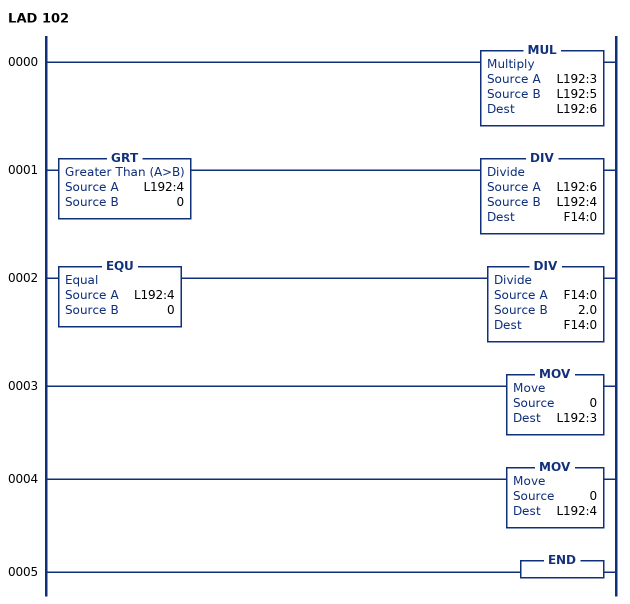
% Rung: 0 %
SOR MUL L192:3 L192:5 L192:6 EOR
% Rung: 1 %
SOR GRT L192:4 0 DIV L192:6 L192:4 F14:0 EOR
% Rung: 2 %
SOR EQU L192:4 0 DIV F14:0 2.0 F14:0 EOR
% Rung: 3 %
SOR MOV 0 L192:3 EOR
% Rung: 4 %
SOR MOV 0 L192:4 EOR
% Rung: 5 %
SOR END EOR

LADDER 103
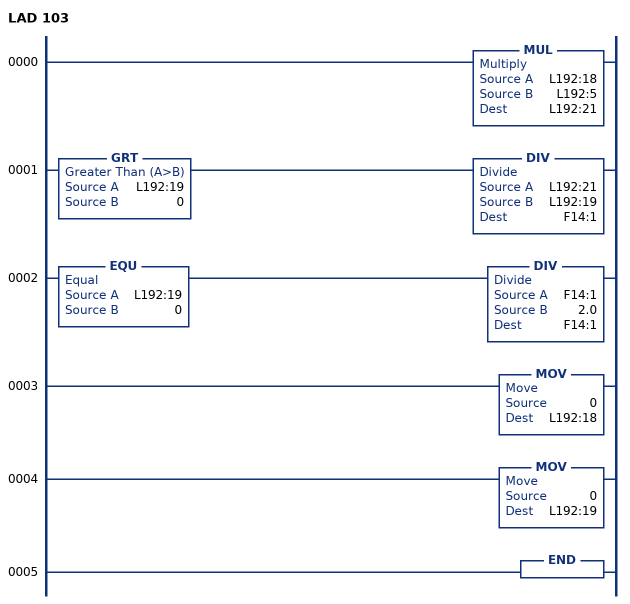
% Rung: 0 %
SOR MUL L192:18 L192:5 L192:21 EOR
% Rung: 1 %
SOR GRT L192:19 0 DIV L192:21 L192:19 F14:1 EOR
% Rung: 2 %
SOR EQU L192:19 0 DIV F14:1 2.0 F14:1 EOR
% Rung: 3 %
SOR MOV 0 L192:18 EOR
% Rung: 4 %
SOR MOV 0 L192:19 EOR
% Rung: 5 %
SOR END EOR

LADDER 104
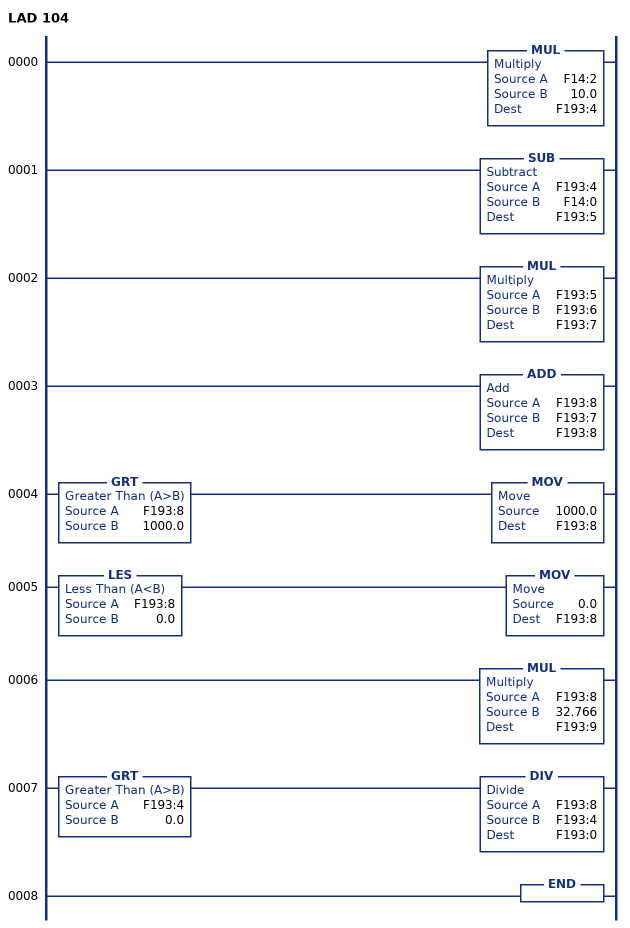
% Rung: 0 %
SOR MUL F14:2 10.0 F193:4 EOR
% Rung: 1 %
SOR SUB F193:4 F14:0 F193:5 EOR
% Rung: 2 %
SOR MUL F193:5 F193:6 F193:7 EOR
% Rung: 3 %
SOR ADD F193:8 F193:7 F193:8 EOR
% Rung: 4 %
SOR GRT F193:8 1000.0 MOV 1000.0 F193:8 EOR
% Rung: 5 %
SOR LES F193:8 0.0 MOV 0.0 F193:8 EOR
% Rung: 6 %
SOR MUL F193:8 32.766 F193:9 EOR
% Rung: 7 %
SOR GRT F193:4 0.0 DIV F193:8 F193:4 F193:0 EOR
% Rung: 8 %
SOR END EOR

LADDER 105
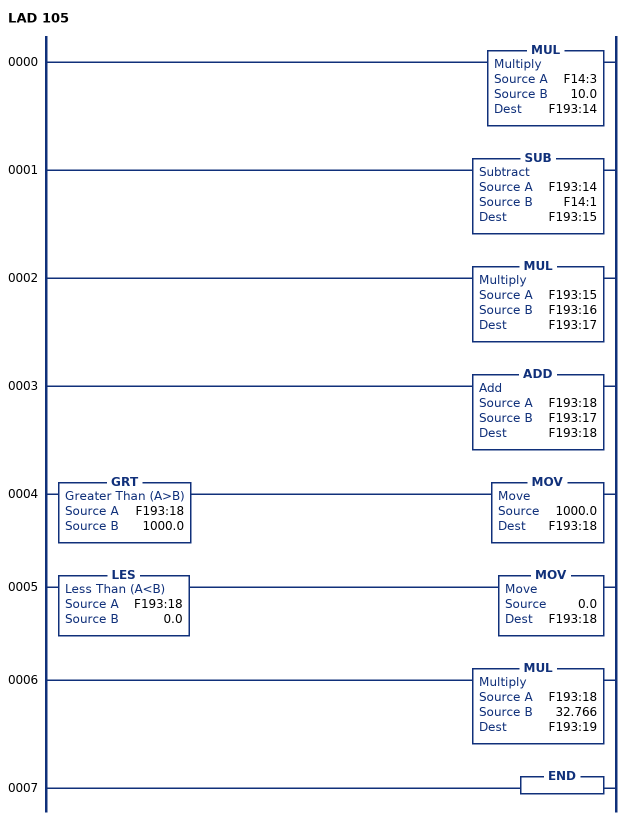
% Rung: 0 %
SOR MUL F14:3 10.0 F193:14 EOR
% Rung: 1 %
SOR SUB F193:14 F14:1 F193:15 EOR
% Rung: 2 %
SOR MUL F193:15 F193:16 F193:17 EOR
% Rung: 3 %
SOR ADD F193:18 F193:17 F193:18 EOR
% Rung: 4 %
SOR GRT F193:18 1000.0 MOV 1000.0 F193:18 EOR
% Rung: 5 %
SOR LES F193:18 0.0 MOV 0.0 F193:18 EOR
% Rung: 6 %
SOR MUL F193:18 32.766 F193:19 EOR
% Rung: 7 %
SOR END EOR

LADDER 110
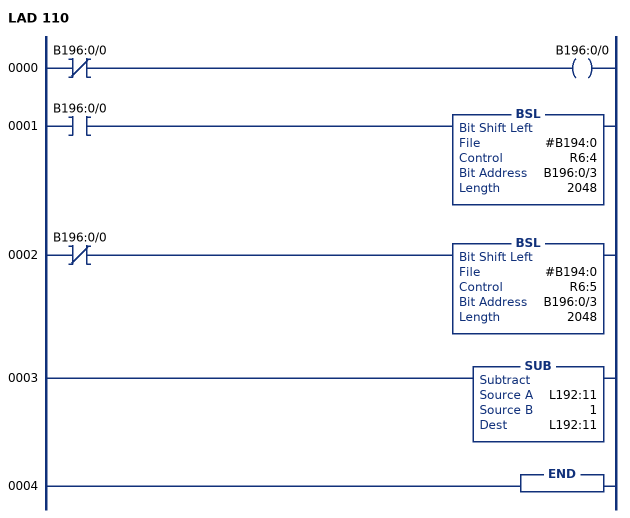
% Rung: 0 %
SOR XIO B196:0/0 OTE B196:0/0 EOR
% Rung: 1 %
SOR XIC B196:0/0 BSL #B194:0 R6:4 B196:0/3 2048 EOR
% Rung: 2 %
SOR XIO B196:0/0 BSL #B194:0 R6:5 B196:0/3 2048 EOR
% Rung: 3 %
SOR SUB L192:11 1 L192:11 EOR
% Rung: 4 %
SOR END EOR

LADDER 111
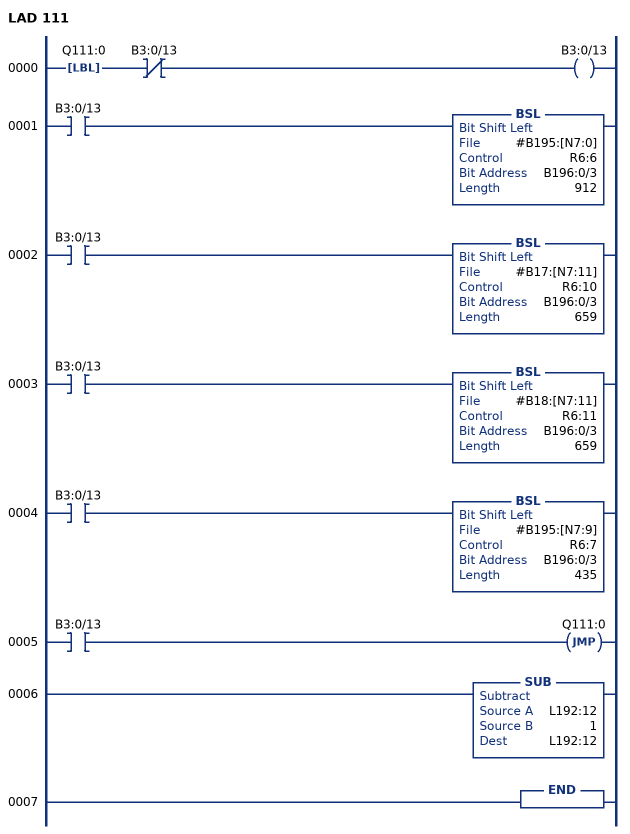
% Rung: 0 %
SOR LBL Q111:0 XIO B3:0/13 OTE B3:0/13 EOR
% Rung: 1 %
SOR XIC B3:0/13 BSL #B195:[N7:0] R6:6 B196:0/3 912 EOR
% Rung: 2 %
SOR XIC B3:0/13 BSL #B17:[N7:11] R6:10 B196:0/3 659 EOR
% Rung: 3 %
SOR XIC B3:0/13 BSL #B18:[N7:11] R6:11 B196:0/3 659 EOR
% Rung: 4 %
SOR XIC B3:0/13 BSL #B195:[N7:9] R6:7 B196:0/3 435 EOR
% Rung: 5 %
SOR XIC B3:0/13 JMP Q111:0 EOR
% Rung: 6 %
SOR SUB L192:12 1 L192:12 EOR
% Rung: 7 %
SOR END EOR

LADDER 122
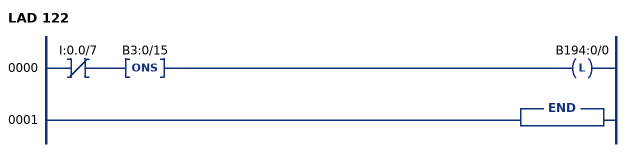
% Rung: 0 %
SOR XIO I:0.0/7 ONS B3:0/15 OTL B194:0/0 EOR
% Rung: 1 %
SOR END EOR

LADDER 125
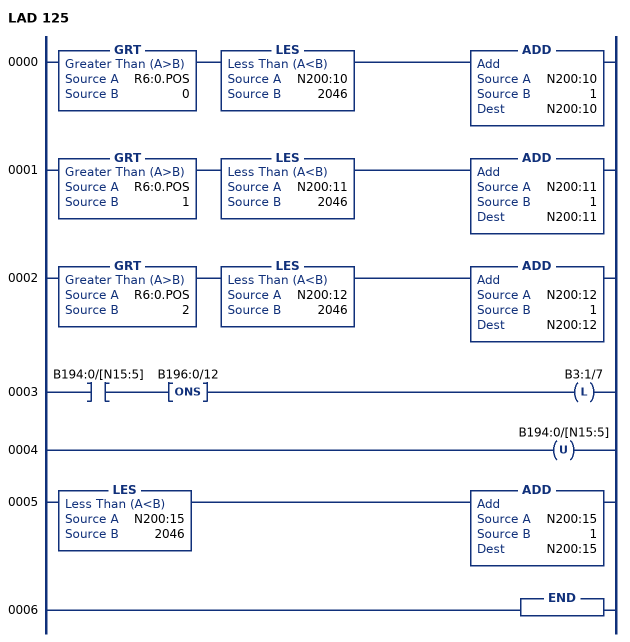
% Rung: 0 %
SOR GRT R6:0.POS 0 LES N200:10 2046 ADD N200:10 1 N200:10 EOR
% Rung: 1 %
SOR GRT R6:0.POS 1 LES N200:11 2046 ADD N200:11 1 N200:11 EOR
% Rung: 2 %
SOR GRT R6:0.POS 2 LES N200:12 2046 ADD N200:12 1 N200:12 EOR
% Rung: 3 %
SOR XIC B194:0/[N15:5] ONS B196:0/12 OTL B3:1/7 EOR
% Rung: 4 %
SOR OTU B194:0/[N15:5] EOR
% Rung: 5 %
SOR LES N200:15 2046 ADD N200:15 1 N200:15 EOR
% Rung: 6 %
SOR END EOR

LADDER 126
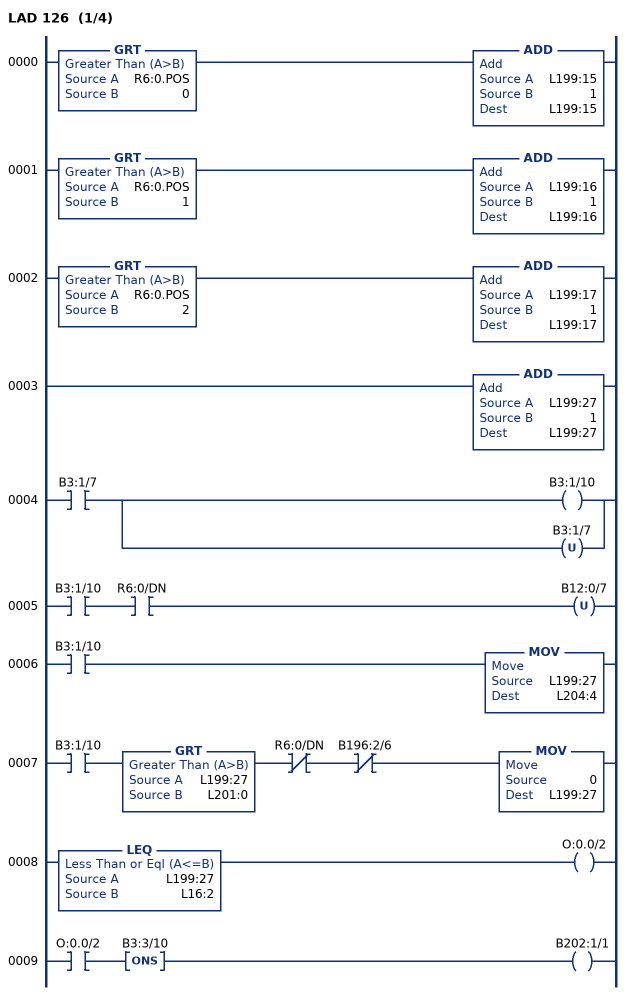
% Rung: 0 %
SOR GRT R6:0.POS 0 ADD L199:15 1 L199:15 EOR
% Rung: 1 %
SOR GRT R6:0.POS 1 ADD L199:16 1 L199:16 EOR
% Rung: 2 %
SOR GRT R6:0.POS 2 ADD L199:17 1 L199:17 EOR
% Rung: 3 %
SOR ADD L199:27 1 L199:27 EOR
% Rung: 4 %
SOR XIC B3:1/7 BST OTE B3:1/10 NXB OTU B3:1/7 BND EOR
% Rung: 5 %
SOR XIC B3:1/10 XIC R6:0/DN OTU B12:0/7 EOR
% Rung: 6 %
SOR XIC B3:1/10 MOV L199:27 L204:4 EOR
% Rung: 7 %
SOR XIC B3:1/10 GRT L199:27 L201:0 XIO R6:0/DN XIO B196:2/6 MOV 0 L199:27 EOR
% Rung: 8 %
SOR LEQ L199:27 L16:2 OTE O:0.0/2 EOR
% Rung: 9 %
SOR XIC O:0.0/2 ONS B3:3/10 OTE B202:1/1 EOR

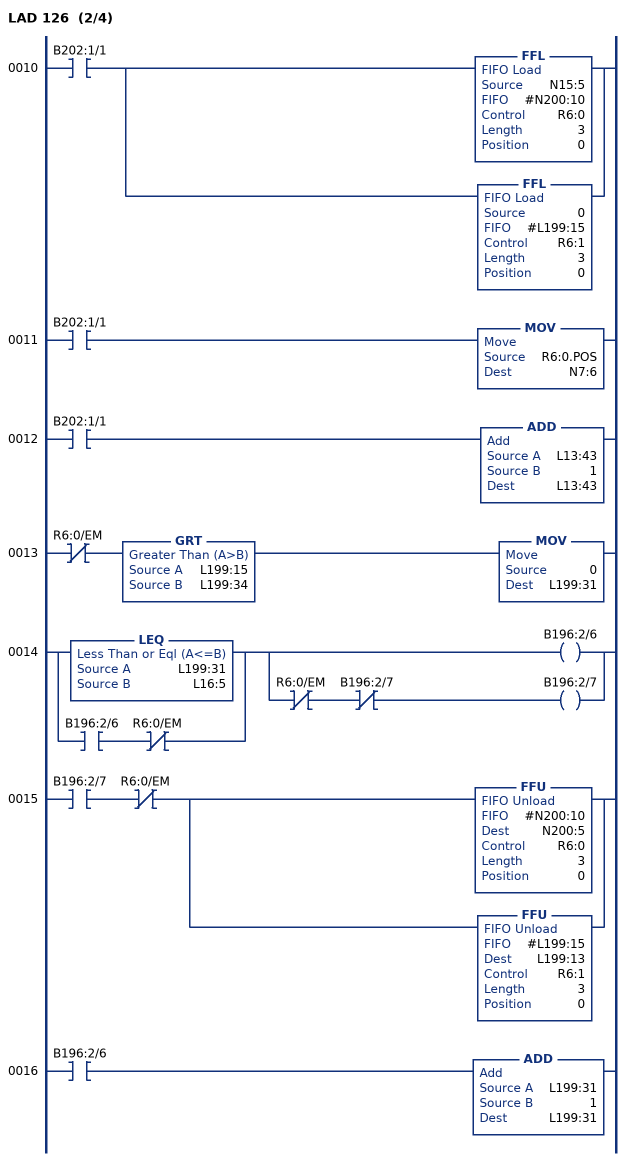
% Rung: 10 %
SOR XIC B202:1/1 BST FFL N15:5 #N200:10 R6:0 3 0 NXB FFL 0 #L199:15 R6:1 3 0 BND EOR
% Rung: 11 %
SOR XIC B202:1/1 MOV R6:0.POS N7:6 EOR
% Rung: 12 %
SOR XIC B202:1/1 ADD L13:43 1 L13:43 EOR
% Rung: 13 %
SOR XIO R6:0/EM GRT L199:15 L199:34 MOV 0 L199:31 EOR
% Rung: 14 %
SOR BST LEQ L199:31 L16:5 NXB XIC B196:2/6 XIO R6:0/EM BND BST OTE B196:2/6 NXB XIO R6:0/EM XIO B196:2/7 OTE B196:2/7 BND EOR
% Rung: 15 %
SOR XIC B196:2/7 XIO R6:0/EM BST FFU #N200:10 N200:5 R6:0 3 0 NXB FFU #L199:15 L199:13 R6:1 3 0 BND EOR
% Rung: 16 %
SOR XIC B196:2/6 ADD L199:31 1 L199:31 EOR

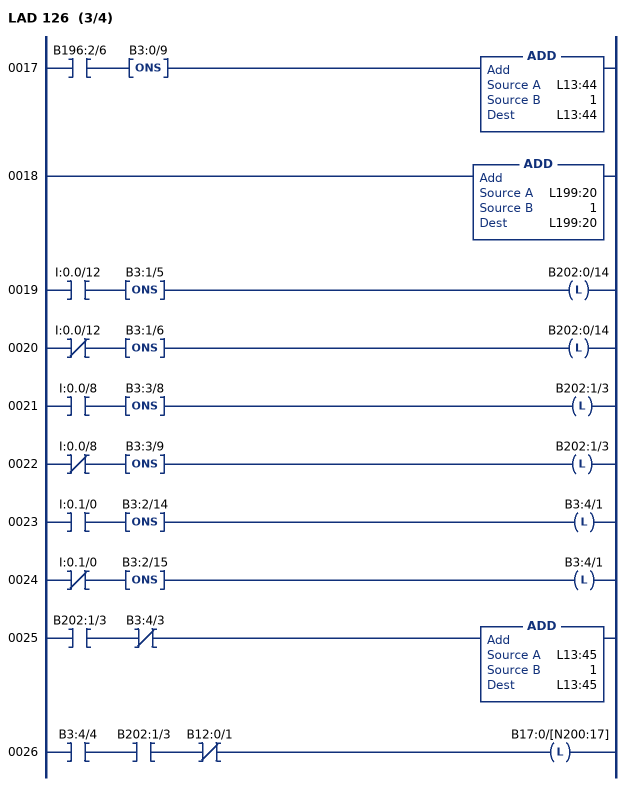
% Rung: 17 %
SOR XIC B196:2/6 ONS B3:0/9 ADD L13:44 1 L13:44 EOR
% Rung: 18 %
SOR ADD L199:20 1 L199:20 EOR
% Rung: 19 %
SOR XIC I:0.0/12 ONS B3:1/5 OTL B202:0/14 EOR
% Rung: 20 %
SOR XIO I:0.0/12 ONS B3:1/6 OTL B202:0/14 EOR
% Rung: 21 %
SOR XIC I:0.0/8 ONS B3:3/8 OTL B202:1/3 EOR
% Rung: 22 %
SOR XIO I:0.0/8 ONS B3:3/9 OTL B202:1/3 EOR
% Rung: 23 %
SOR XIC I:0.1/0 ONS B3:2/14 OTL B3:4/1 EOR
% Rung: 24 %
SOR XIO I:0.1/0 ONS B3:2/15 OTL B3:4/1 EOR
% Rung: 25 %
SOR XIC B202:1/3 XIO B3:4/3 ADD L13:45 1 L13:45 EOR
% Rung: 26 %
SOR XIC B3:4/4 XIC B202:1/3 XIO B12:0/1 OTL B17:0/[N200:17] EOR

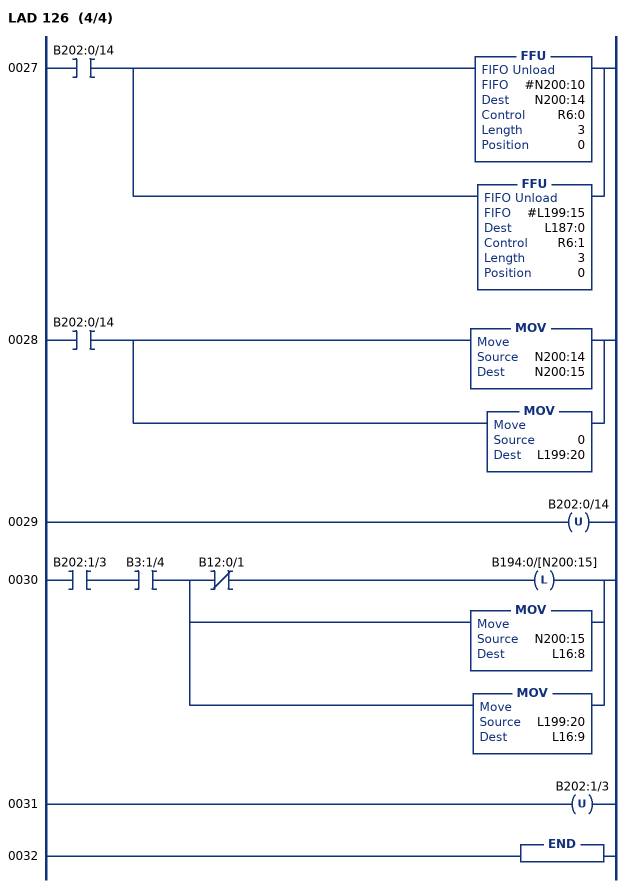
% Rung: 27 %
SOR XIC B202:0/14 BST FFU #N200:10 N200:14 R6:0 3 0 NXB FFU #L199:15 L187:0 R6:1 3 0 BND EOR
% Rung: 28 %
SOR XIC B202:0/14 BST MOV N200:14 N200:15 NXB MOV 0 L199:20 BND EOR
% Rung: 29 %
SOR OTU B202:0/14 EOR
% Rung: 30 %
SOR XIC B202:1/3 XIC B3:1/4 BST XIO B12:0/1 OTL B194:0/[N200:15] NXB MOV N200:15 L16:8 NXB MOV L199:20 L16:9 BND EOR
% Rung: 31 %
SOR OTU B202:1/3 EOR
% Rung: 32 %
SOR END EOR

LADDER 131
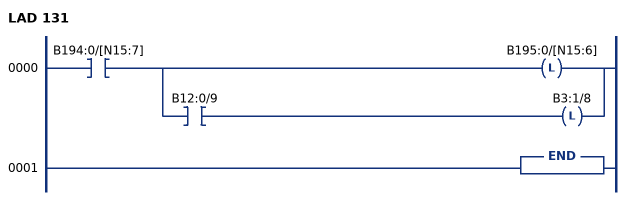
% Rung: 0 %
SOR XIC B194:0/[N15:7] BST OTL B195:0/[N15:6] NXB XIC B12:0/9 OTL B3:1/8 BND EOR
% Rung: 1 %
SOR END EOR

LADDER 141
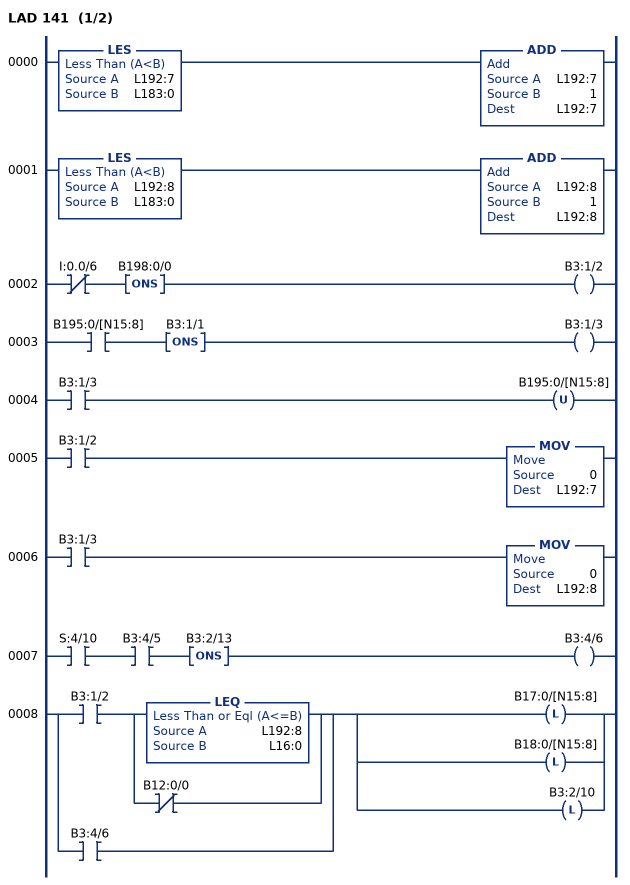
% Rung: 0 %
SOR LES L192:7 L183:0 ADD L192:7 1 L192:7 EOR
% Rung: 1 %
SOR LES L192:8 L183:0 ADD L192:8 1 L192:8 EOR
% Rung: 2 %
SOR XIO I:0.0/6 ONS B198:0/0 OTE B3:1/2 EOR
% Rung: 3 %
SOR XIC B195:0/[N15:8] ONS B3:1/1 OTE B3:1/3 EOR
% Rung: 4 %
SOR XIC B3:1/3 OTU B195:0/[N15:8] EOR
% Rung: 5 %
SOR XIC B3:1/2 MOV 0 L192:7 EOR
% Rung: 6 %
SOR XIC B3:1/3 MOV 0 L192:8 EOR
% Rung: 7 %
SOR XIC S:4/10 XIC B3:4/5 ONS B3:2/13 OTE B3:4/6 EOR
% Rung: 8 %
SOR BST XIC B3:1/2 BST LEQ L192:8 L16:0 NXB XIO B12:0/0 BND NXB XIC B3:4/6 BND BST OTL B17:0/[N15:8] NXB OTL B18:0/[N15:8] NXB OTL B3:2/10 BND EOR

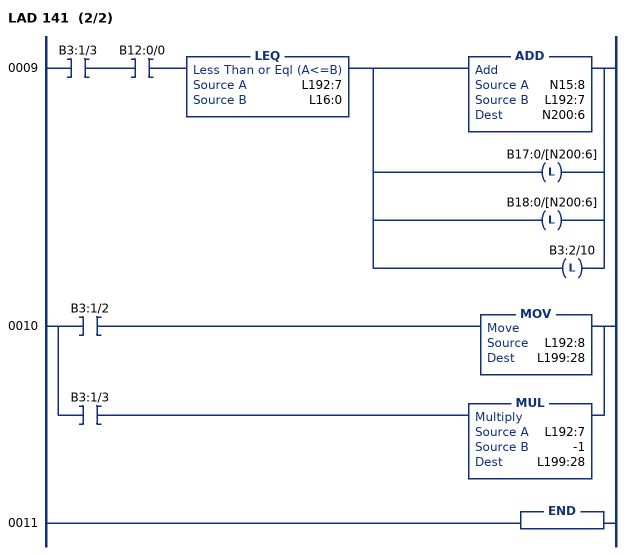
% Rung: 9 %
SOR XIC B3:1/3 XIC B12:0/0 LEQ L192:7 L16:0 BST ADD N15:8 L192:7 N200:6 NXB OTL B17:0/[N200:6] NXB OTL B18:0/[N200:6] NXB OTL B3:2/10 BND EOR
% Rung: 10 %
SOR BST XIC B3:1/2 MOV L192:8 L199:28 NXB XIC B3:1/3 MUL L192:7 -1 L199:28 BND EOR
% Rung: 11 %
SOR END EOR

LADDER 150
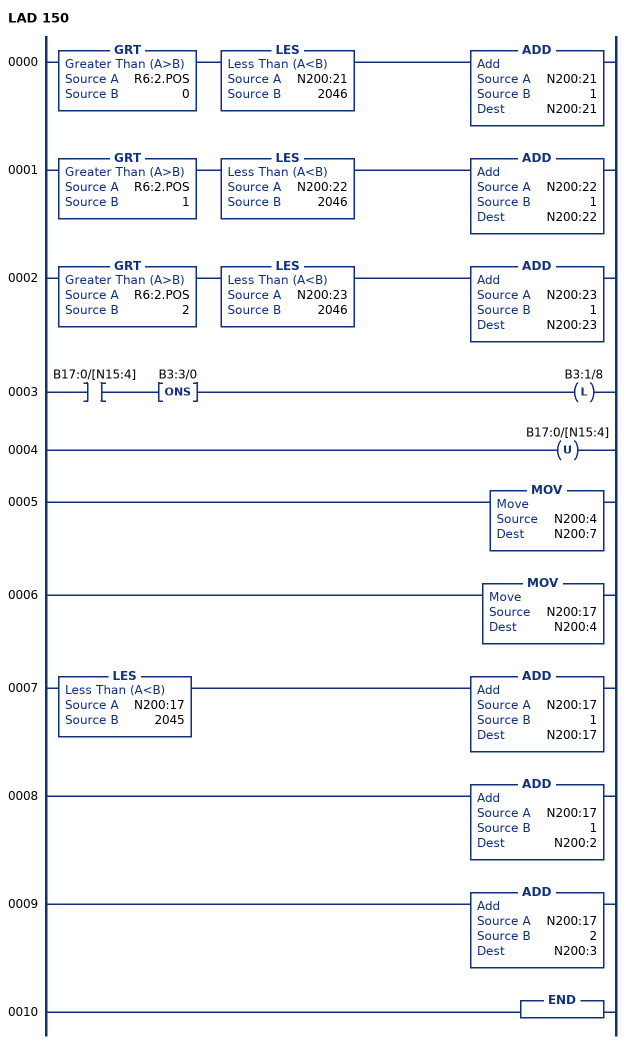
% Rung: 0 %
SOR GRT R6:2.POS 0 LES N200:21 2046 ADD N200:21 1 N200:21 EOR
% Rung: 1 %
SOR GRT R6:2.POS 1 LES N200:22 2046 ADD N200:22 1 N200:22 EOR
% Rung: 2 %
SOR GRT R6:2.POS 2 LES N200:23 2046 ADD N200:23 1 N200:23 EOR
% Rung: 3 %
SOR XIC B17:0/[N15:4] ONS B3:3/0 OTL B3:1/8 EOR
% Rung: 4 %
SOR OTU B17:0/[N15:4] EOR
% Rung: 5 %
SOR MOV N200:4 N200:7 EOR
% Rung: 6 %
SOR MOV N200:17 N200:4 EOR
% Rung: 7 %
SOR LES N200:17 2045 ADD N200:17 1 N200:17 EOR
% Rung: 8 %
SOR ADD N200:17 1 N200:2 EOR
% Rung: 9 %
SOR ADD N200:17 2 N200:3 EOR
% Rung: 10 %
SOR END EOR

LADDER 151
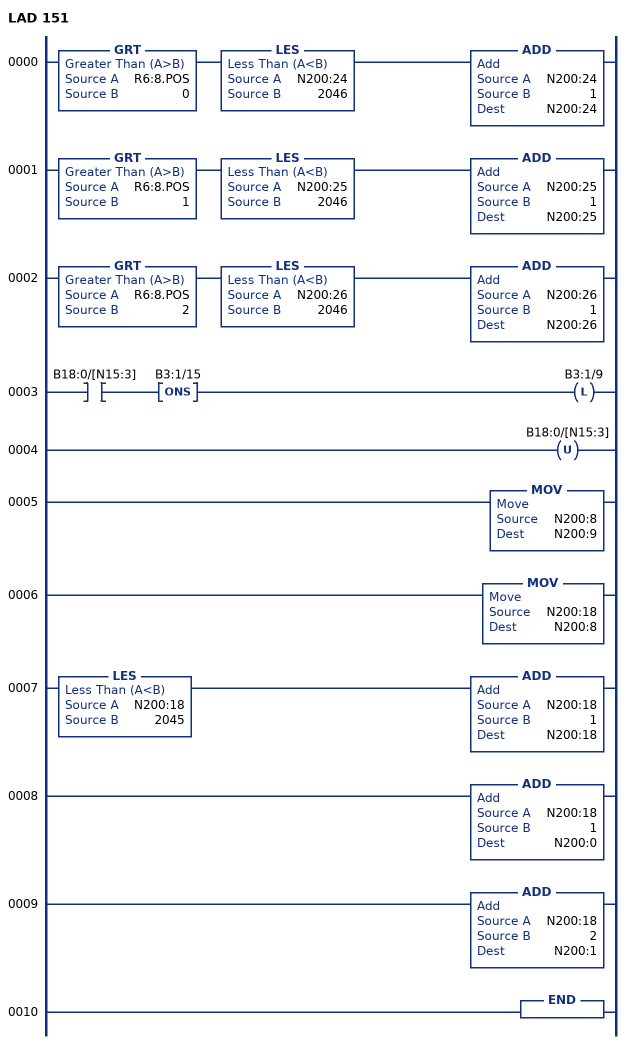
% Rung: 0 %
SOR GRT R6:8.POS 0 LES N200:24 2046 ADD N200:24 1 N200:24 EOR
% Rung: 1 %
SOR GRT R6:8.POS 1 LES N200:25 2046 ADD N200:25 1 N200:25 EOR
% Rung: 2 %
SOR GRT R6:8.POS 2 LES N200:26 2046 ADD N200:26 1 N200:26 EOR
% Rung: 3 %
SOR XIC B18:0/[N15:3] ONS B3:1/15 OTL B3:1/9 EOR
% Rung: 4 %
SOR OTU B18:0/[N15:3] EOR
% Rung: 5 %
SOR MOV N200:8 N200:9 EOR
% Rung: 6 %
SOR MOV N200:18 N200:8 EOR
% Rung: 7 %
SOR LES N200:18 2045 ADD N200:18 1 N200:18 EOR
% Rung: 8 %
SOR ADD N200:18 1 N200:0 EOR
% Rung: 9 %
SOR ADD N200:18 2 N200:1 EOR
% Rung: 10 %
SOR END EOR

LADDER 160
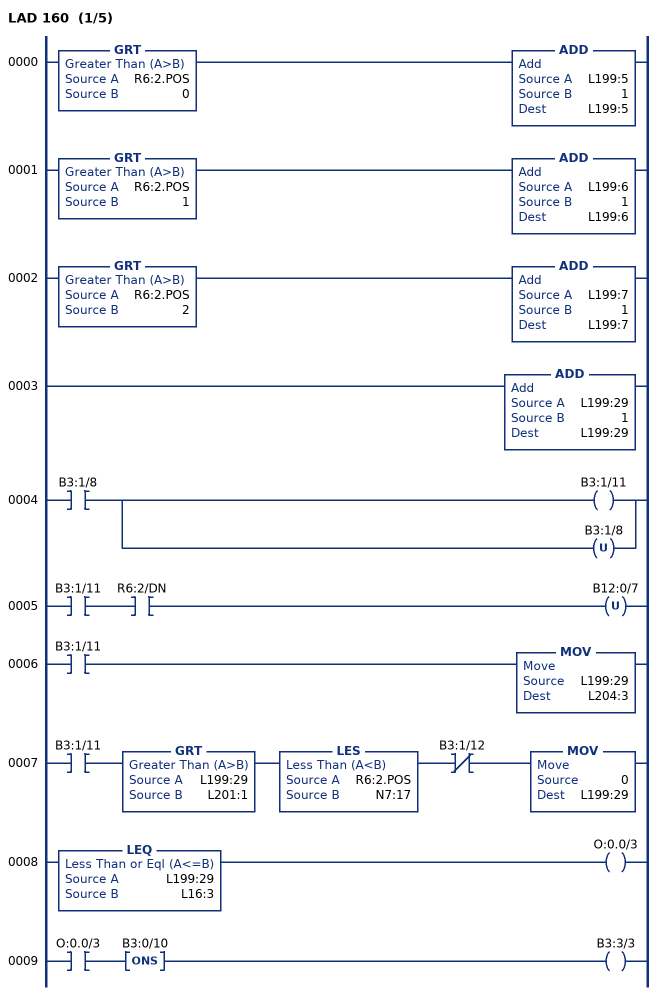
% Rung: 0 %
SOR GRT R6:2.POS 0 ADD L199:5 1 L199:5 EOR
% Rung: 1 %
SOR GRT R6:2.POS 1 ADD L199:6 1 L199:6 EOR
% Rung: 2 %
SOR GRT R6:2.POS 2 ADD L199:7 1 L199:7 EOR
% Rung: 3 %
SOR ADD L199:29 1 L199:29 EOR
% Rung: 4 %
SOR XIC B3:1/8 BST OTE B3:1/11 NXB OTU B3:1/8 BND EOR
% Rung: 5 %
SOR XIC B3:1/11 XIC R6:2/DN OTU B12:0/7 EOR
% Rung: 6 %
SOR XIC B3:1/11 MOV L199:29 L204:3 EOR
% Rung: 7 %
SOR XIC B3:1/11 GRT L199:29 L201:1 LES R6:2.POS N7:17 XIO B3:1/12 MOV 0 L199:29 EOR
% Rung: 8 %
SOR LEQ L199:29 L16:3 OTE O:0.0/3 EOR
% Rung: 9 %
SOR XIC O:0.0/3 ONS B3:0/10 OTE B3:3/3 EOR

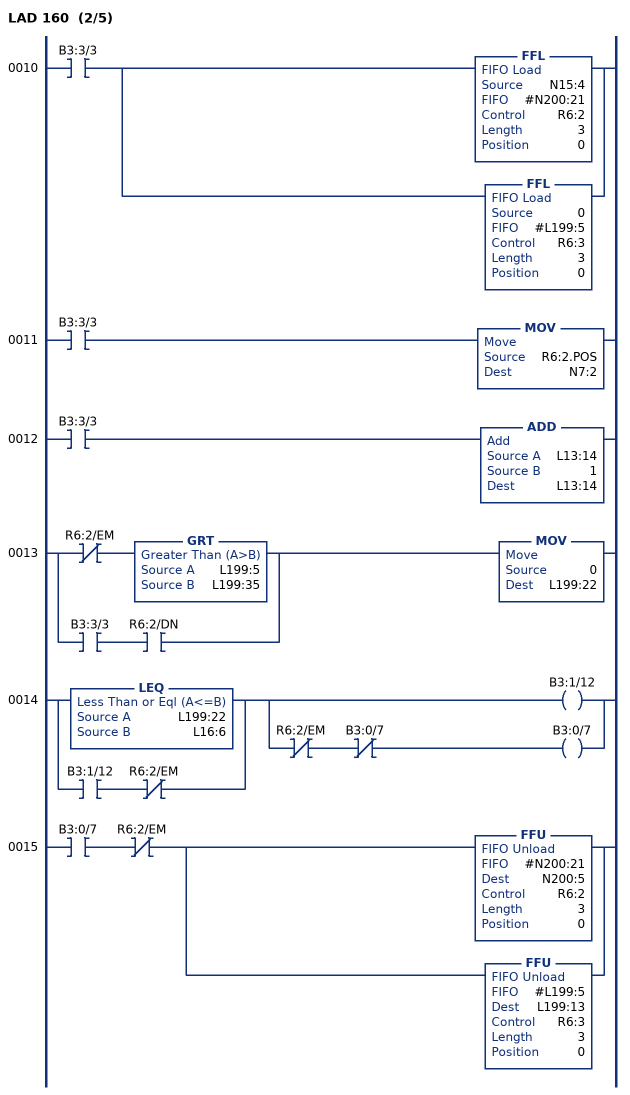
% Rung: 10 %
SOR XIC B3:3/3 BST FFL N15:4 #N200:21 R6:2 3 0 NXB FFL 0 #L199:5 R6:3 3 0 BND EOR
% Rung: 11 %
SOR XIC B3:3/3 MOV R6:2.POS N7:2 EOR
% Rung: 12 %
SOR XIC B3:3/3 ADD L13:14 1 L13:14 EOR
% Rung: 13 %
SOR BST XIO R6:2/EM GRT L199:5 L199:35 NXB XIC B3:3/3 XIC R6:2/DN BND MOV 0 L199:22 EOR
% Rung: 14 %
SOR BST LEQ L199:22 L16:6 NXB XIC B3:1/12 XIO R6:2/EM BND BST OTE B3:1/12 NXB XIO R6:2/EM XIO B3:0/7 OTE B3:0/7 BND EOR
% Rung: 15 %
SOR XIC B3:0/7 XIO R6:2/EM BST FFU #N200:21 N200:5 R6:2 3 0 NXB FFU #L199:5 L199:13 R6:3 3 0 BND EOR

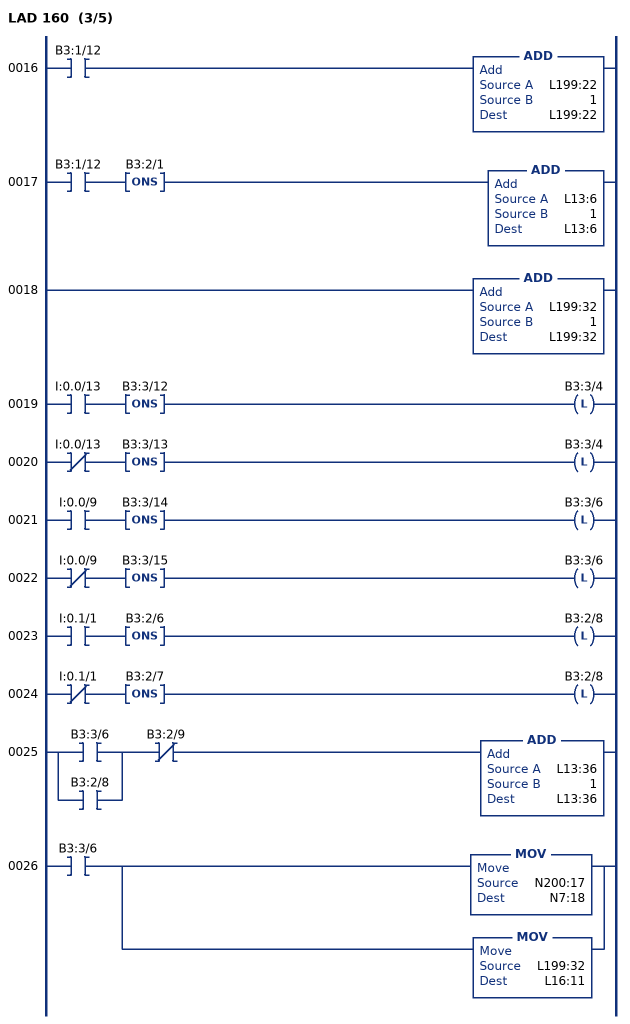
% Rung: 16 %
SOR XIC B3:1/12 ADD L199:22 1 L199:22 EOR
% Rung: 17 %
SOR XIC B3:1/12 ONS B3:2/1 ADD L13:6 1 L13:6 EOR
% Rung: 18 %
SOR ADD L199:32 1 L199:32 EOR
% Rung: 19 %
SOR XIC I:0.0/13 ONS B3:3/12 OTL B3:3/4 EOR
% Rung: 20 %
SOR XIO I:0.0/13 ONS B3:3/13 OTL B3:3/4 EOR
% Rung: 21 %
SOR XIC I:0.0/9 ONS B3:3/14 OTL B3:3/6 EOR
% Rung: 22 %
SOR XIO I:0.0/9 ONS B3:3/15 OTL B3:3/6 EOR
% Rung: 23 %
SOR XIC I:0.1/1 ONS B3:2/6 OTL B3:2/8 EOR
% Rung: 24 %
SOR XIO I:0.1/1 ONS B3:2/7 OTL B3:2/8 EOR
% Rung: 25 %
SOR BST XIC B3:3/6 NXB XIC B3:2/8 BND XIO B3:2/9 ADD L13:36 1 L13:36 EOR
% Rung: 26 %
SOR XIC B3:3/6 BST MOV N200:17 N7:18 NXB MOV L199:32 L16:11 BND EOR

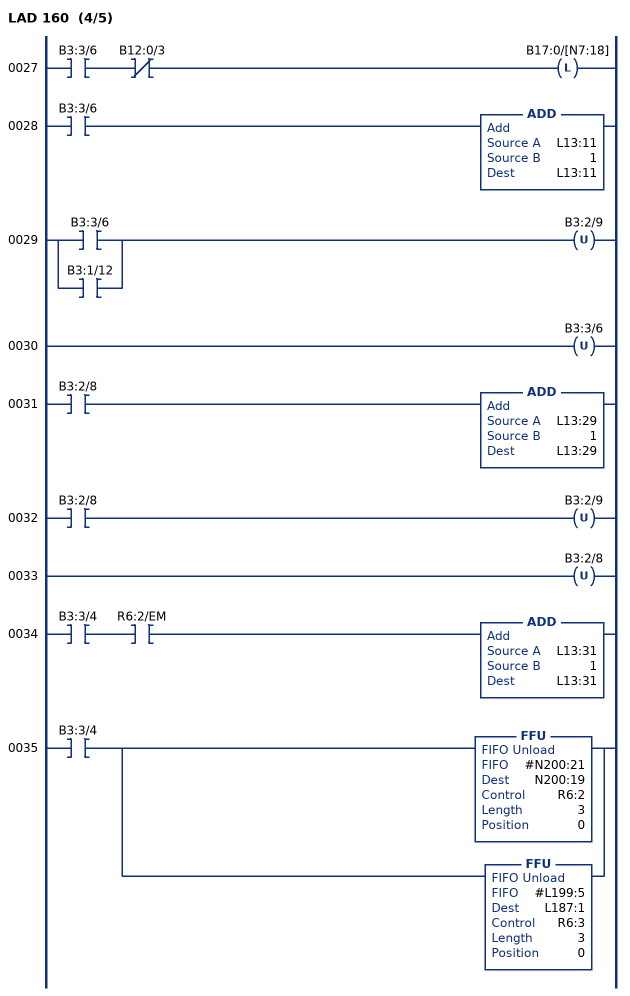
% Rung: 27 %
SOR XIC B3:3/6 XIO B12:0/3 OTL B17:0/[N7:18] EOR
% Rung: 28 %
SOR XIC B3:3/6 ADD L13:11 1 L13:11 EOR
% Rung: 29 %
SOR BST XIC B3:3/6 NXB XIC B3:1/12 BND OTU B3:2/9 EOR
% Rung: 30 %
SOR OTU B3:3/6 EOR
% Rung: 31 %
SOR XIC B3:2/8 ADD L13:29 1 L13:29 EOR
% Rung: 32 %
SOR XIC B3:2/8 OTU B3:2/9 EOR
% Rung: 33 %
SOR OTU B3:2/8 EOR
% Rung: 34 %
SOR XIC B3:3/4 XIC R6:2/EM ADD L13:31 1 L13:31 EOR
% Rung: 35 %
SOR XIC B3:3/4 BST FFU #N200:21 N200:19 R6:2 3 0 NXB FFU #L199:5 L187:1 R6:3 3 0 BND EOR

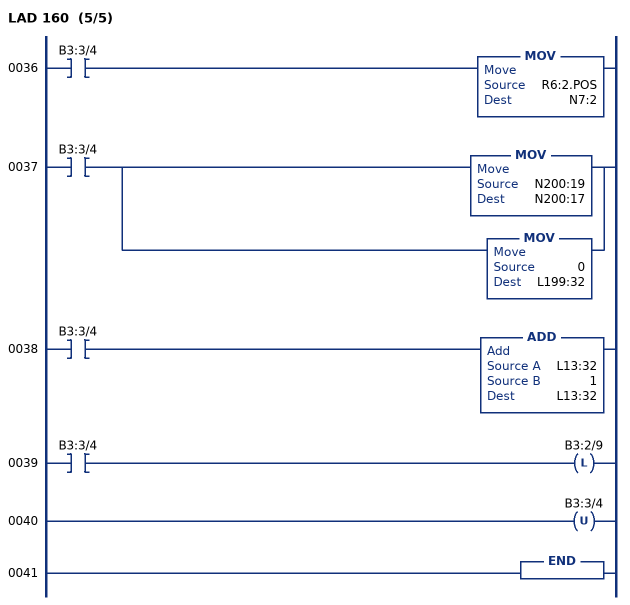
% Rung: 36 %
SOR XIC B3:3/4 MOV R6:2.POS N7:2 EOR
% Rung: 37 %
SOR XIC B3:3/4 BST MOV N200:19 N200:17 NXB MOV 0 L199:32 BND EOR
% Rung: 38 %
SOR XIC B3:3/4 ADD L13:32 1 L13:32 EOR
% Rung: 39 %
SOR XIC B3:3/4 OTL B3:2/9 EOR
% Rung: 40 %
SOR OTU B3:3/4 EOR
% Rung: 41 %
SOR END EOR

LADDER 161
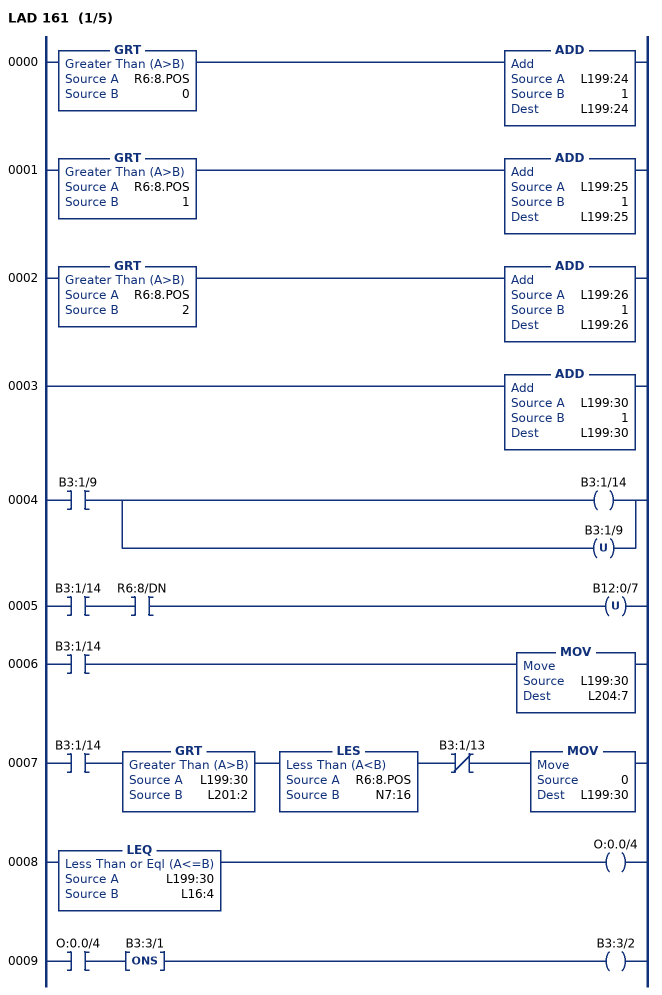
% Rung: 0 %
SOR GRT R6:8.POS 0 ADD L199:24 1 L199:24 EOR
% Rung: 1 %
SOR GRT R6:8.POS 1 ADD L199:25 1 L199:25 EOR
% Rung: 2 %
SOR GRT R6:8.POS 2 ADD L199:26 1 L199:26 EOR
% Rung: 3 %
SOR ADD L199:30 1 L199:30 EOR
% Rung: 4 %
SOR XIC B3:1/9 BST OTE B3:1/14 NXB OTU B3:1/9 BND EOR
% Rung: 5 %
SOR XIC B3:1/14 XIC R6:8/DN OTU B12:0/7 EOR
% Rung: 6 %
SOR XIC B3:1/14 MOV L199:30 L204:7 EOR
% Rung: 7 %
SOR XIC B3:1/14 GRT L199:30 L201:2 LES R6:8.POS N7:16 XIO B3:1/13 MOV 0 L199:30 EOR
% Rung: 8 %
SOR LEQ L199:30 L16:4 OTE O:0.0/4 EOR
% Rung: 9 %
SOR XIC O:0.0/4 ONS B3:3/1 OTE B3:3/2 EOR

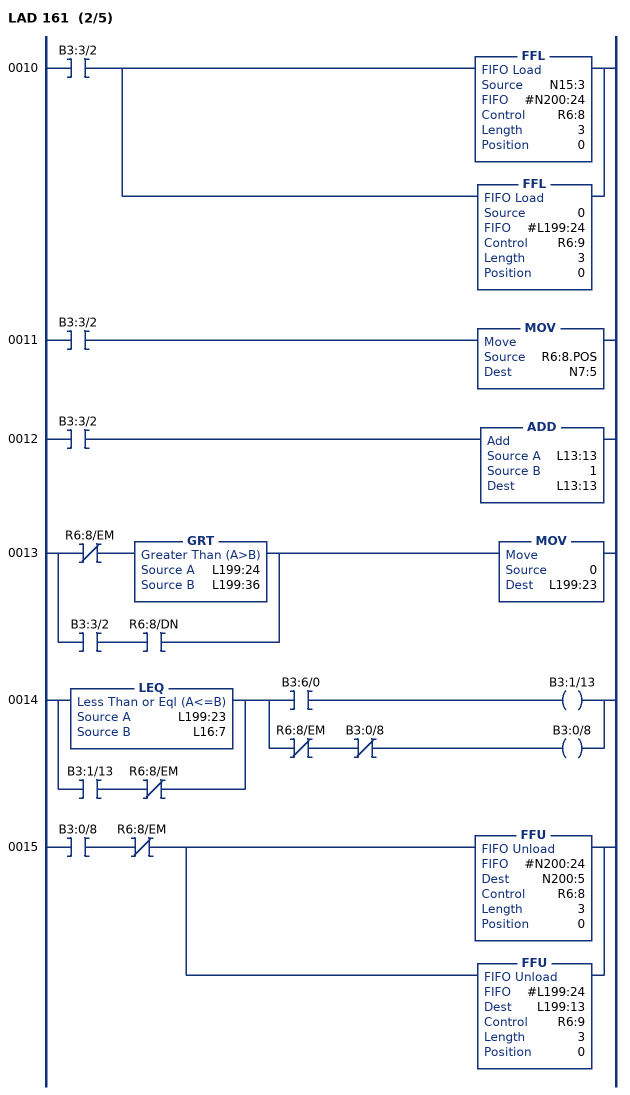
% Rung: 10 %
SOR XIC B3:3/2 BST FFL N15:3 #N200:24 R6:8 3 0 NXB FFL 0 #L199:24 R6:9 3 0 BND EOR
% Rung: 11 %
SOR XIC B3:3/2 MOV R6:8.POS N7:5 EOR
% Rung: 12 %
SOR XIC B3:3/2 ADD L13:13 1 L13:13 EOR
% Rung: 13 %
SOR BST XIO R6:8/EM GRT L199:24 L199:36 NXB XIC B3:3/2 XIC R6:8/DN BND MOV 0 L199:23 EOR
% Rung: 14 %
SOR BST LEQ L199:23 L16:7 NXB XIC B3:1/13 XIO R6:8/EM BND BST XIC B3:6/0 OTE B3:1/13 NXB XIO R6:8/EM XIO B3:0/8 OTE B3:0/8 BND EOR
% Rung: 15 %
SOR XIC B3:0/8 XIO R6:8/EM BST FFU #N200:24 N200:5 R6:8 3 0 NXB FFU #L199:24 L199:13 R6:9 3 0 BND EOR

